FUNCTION_BLOCK FB_SampleListener EXTENDS FB_ListenerBase2
VAR_INPUT
END_VAR
VAR_OUTPUT
END_VAR
VAR
	sJsonAttribute : STRING (10000);	
	hr : HRESULT;
	
	nCntMessagesSent : INT;
	nCntAlarmsRaised : INT;
	nCntAlarmsConfirmed : INT;
	nCntAlarmsCleared : INT;
	
	//text retrieval of message
	fbRequestEventText : FB_RequestEventText;
	{attribute 'TcEncoding':='UTF-8'}
	sLastMessageText : STRING;
	bReqText : BOOL;
END_VAR

METHOD Execute : HRESULT
VAR_INPUT
END_VAR
Execute := SUPER^.Execute(); //retrieve events

//retrieve the text of a message
IF 	bReqText AND fbRequestEventText.bError THEN 
	sLastMessageText := 'Error';
	bReqText := FALSE; 
ELSIF bReqText AND NOT  fbRequestEventText.bBusy THEN
	fbRequestEventText.GetString(sLastMessageText, SIZEOF(sLastMessageText));
	bReqText := FALSE;
END_IF
END_METHOD

METHOD OnAlarmCleared : HRESULT
VAR_INPUT
	fbEvent : REFERENCE TO FB_TcEvent;
END_VAR
nCntAlarmsCleared := nCntAlarmsCleared + 1;

OnAlarmCleared := S_OK; // in order to receive more callbacks (Set <> S_OK in order to cancel the callbacks for this program cycle.)
END_METHOD

METHOD OnAlarmConfirmed : HRESULT
VAR_INPUT
	fbEvent : REFERENCE TO FB_TcEvent;
END_VAR
nCntAlarmsConfirmed := nCntAlarmsConfirmed + 1;

OnAlarmConfirmed := S_OK; // in order to receive more callbacks (Set <> S_OK in order to cancel the callbacks for this program cycle.)
END_METHOD

METHOD OnAlarmRaised : HRESULT
VAR_INPUT
	fbEvent : REFERENCE TO FB_TcEvent;
END_VAR
hr := fbEvent.GetJsonAttribute(sJsonAttribute, SIZEOF(sJsonAttribute));
nCntAlarmsRaised := nCntAlarmsRaised + 1;

OnAlarmRaised := S_OK; // in order to receive more callbacks (Set <> S_OK in order to cancel the callbacks for this program cycle.)
END_METHOD

METHOD OnMessageSent : HRESULT
VAR_INPUT
	fbEvent : REFERENCE TO FB_TcEvent;
END_VAR

VAR 
END_VAR
hr := fbEvent.GetJsonAttribute(sJsonAttribute, SIZEOF(sJsonAttribute));
nCntMessagesSent := nCntMessagesSent + 1;

fbRequestEventText.Request(eventClass:=fbEvent.EventClass, nEventId:=fbEvent.nEventId, nLangId:=TcLcid.en_US, ipArgs:=fbEvent.ipArguments );
bReqText := TRUE;

OnMessageSent := S_OK; // in order to receive more callbacks (Set <> S_OK in order to cancel the callbacks for this program cycle.)
END_METHOD

END_FUNCTION_BLOCK

(* stored: Version 1.1.0.1, ProductVersion 3.1.4024.12
   POU FB_SampleListener: Id {50ed088d-9a7d-4c16-86a9-e90b487e4982}, SpecialFunc None
   Method Execute: Id {3c7f655d-2c73-41dc-b085-26c5a3b1cef1}
   Method OnAlarmCleared: Id {036602cd-44fc-40d2-99e6-e6b033452290}
   Method OnAlarmConfirmed: Id {efe870ed-8bbd-4c42-9405-bf33d81f12d4}
   Method OnAlarmRaised: Id {1df5b803-888d-4d2d-ab12-93687f9c1a1e}
   Method OnMessageSent: Id {b4dac56d-cfe9-4434-ae5b-afa117054bdb} *)
